// TIA Portal V20 export
TYPE "typeCmInterfaceSoftCam"
// stored: Access Published, Namespace Unit1.Em6
   STRUCT
      visionUnit : "Unit1.Em6.typeCmInterfaceSoftCamVisionController";
   END_STRUCT;
END_TYPE
